(* IEC 61131-3 sources: RL_MAR/experiments/comparison/llm4plc/results/deepseek-ai-DeepSeek-V3.2_20260506_104945/20260506_124247, 4 files *)

(* ---- generated_code_iteration_0.st ---- *)
START_ST
FUNCTION_BLOCK MultimediaArtInstallationControl
VAR_INPUT
    MotionSensor : BOOL; (* Motion detection input *)
    AudioTrack : BOOL; (* Selected audio track *)
    VisualContent : BOOL; (* Selected visual content *)
END_VAR
VAR_OUTPUT
    LightingControl : BOOL; (* Lighting control output *)
    AudioControl : BOOL; (* Audio playback control *)
    VisualControl : BOOL; (* Visual display control *)
END_VAR
VAR
    ActivationTimer : INT; (* Timer for activation duration *)
    state : INT; (* Current state: 0 = IDLE_WAITING_FOR_MOTION, 1 = ACTIVE_ELEMENTS_ON *)
    prevState : INT; (* Previous state for detecting state changes *)
END_VAR

(* State definitions *)
CONST
    STATE_IDLE := 0;
    STATE_ACTIVE := 1;
END_CONST

(* State machine execution *)
CASE state OF
    STATE_IDLE: (* IDLE_WAITING_FOR_MOTION *)
        (* Set outputs to FALSE *)
        LightingControl := FALSE;
        AudioControl := FALSE;
        VisualControl := FALSE;

        (* Check transition to ACTIVE_ELEMENTS_ON *)
        IF MotionSensor THEN
            (* Reset timer and transition to active state *)
            ActivationTimer := 0;
            state := STATE_ACTIVE;
        END_IF;

    STATE_ACTIVE: (* ACTIVE_ELEMENTS_ON *)
        (* Set outputs to TRUE *)
        LightingControl := TRUE;
        AudioControl := TRUE;
        VisualControl := TRUE;

        (* Increment activation timer each cycle *)
        ActivationTimer := ActivationTimer + 1;

        (* Check transition back to IDLE *)
        IF (NOT MotionSensor) OR (ActivationTimer >= 300) THEN
            (* Reset timer and transition to idle state *)
            ActivationTimer := 0;
            state := STATE_IDLE;
        END_IF;

END_CASE;

(* Store current state for next cycle *)
prevState := state;

END_FUNCTION_BLOCK
END_ST

(* ---- generated_code_iteration_1.st ---- *)
START_REASON
The validation feedback indicates a syntax error in the CODESYS compiler validation. Specifically, it states: "应该用';' 替换'STATE_IDLE'", which translates to "should replace 'STATE_IDLE' with ';'". This suggests that in the CONST section, the constant declaration for STATE_IDLE is missing a semicolon at the end of the line. In Structured Text (ST), constant declarations must end with a semicolon, similar to variable declarations. The current code has "STATE_IDLE := 0;" but the feedback implies it's incorrectly written. However, looking at the provided code, the CONST section is:

CONST
    STATE_IDLE := 0;
    STATE_ACTIVE := 1;
END_CONST

This appears correct with semicolons. But the feedback might be pointing to a deeper issue: in CODESYS, constant declarations in a FUNCTION_BLOCK might require a different syntax or placement. Alternatively, the error could be due to a missing semicolon after "END_CONST" or an issue with the CASE statement. Upon review, the CASE statement uses "STATE_IDLE:" as a label, which is correct. The feedback might be misleading, but to comply, I'll ensure all syntax is correct. Perhaps the CONST section should be inside the VAR block or declared differently. In CODESYS, constants can be declared within the VAR_CONSTANT section. I'll restructure the code to use VAR_CONSTANT instead of CONST for better CODESYS compatibility. Also, I'll verify all semicolons are properly placed.

Additionally, I'll ensure the FUNCTION_BLOCK structure is maintained with proper variable sections closed with END_VAR, not END_VAR_INPUT or END_VAR_OUTPUT. The current code uses END_VAR correctly, but I'll double-check.

The core issue is likely the CONST declaration method. I'll change it to VAR_CONSTANT to align with CODESYS standards.
END_REASON

START_ST
FUNCTION_BLOCK MultimediaArtInstallationControl
VAR_INPUT
    MotionSensor : BOOL; (* Motion detection input *)
    AudioTrack : BOOL; (* Selected audio track *)
    VisualContent : BOOL; (* Selected visual content *)
END_VAR
VAR_OUTPUT
    LightingControl : BOOL; (* Lighting control output *)
    AudioControl : BOOL; (* Audio playback control *)
    VisualControl : BOOL; (* Visual display control *)
END_VAR
VAR
    ActivationTimer : INT; (* Timer for activation duration *)
    state : INT; (* Current state: 0 = IDLE_WAITING_FOR_MOTION, 1 = ACTIVE_ELEMENTS_ON *)
    prevState : INT; (* Previous state for detecting state changes *)
END_VAR
VAR_CONSTANT
    STATE_IDLE : INT := 0;
    STATE_ACTIVE : INT := 1;
END_VAR

(* State machine execution *)
CASE state OF
    STATE_IDLE: (* IDLE_WAITING_FOR_MOTION *)
        (* Set outputs to FALSE *)
        LightingControl := FALSE;
        AudioControl := FALSE;
        VisualControl := FALSE;

        (* Check transition to ACTIVE_ELEMENTS_ON *)
        IF MotionSensor THEN
            (* Reset timer and transition to active state *)
            ActivationTimer := 0;
            state := STATE_ACTIVE;
        END_IF;

    STATE_ACTIVE: (* ACTIVE_ELEMENTS_ON *)
        (* Set outputs to TRUE *)
        LightingControl := TRUE;
        AudioControl := TRUE;
        VisualControl := TRUE;

        (* Increment activation timer each cycle *)
        ActivationTimer := ActivationTimer + 1;

        (* Check transition back to IDLE *)
        IF (NOT MotionSensor) OR (ActivationTimer >= 300) THEN
            (* Reset timer and transition to idle state *)
            ActivationTimer := 0;
            state := STATE_IDLE;
        END_IF;

END_CASE;

(* Store current state for next cycle *)
prevState := state;

END_FUNCTION_BLOCK
END_ST

(* ---- generated_code_iteration_2.st ---- *)
START_REASON
The validation feedback indicates an encoding issue with the CODESYS compiler, specifically: "'gbk' codec can't decode byte 0xaf in position 129: illegal multibyte sequence". This suggests that there are non-ASCII characters in the code that the compiler cannot decode using the GBK encoding. The most likely source is the Chinese comments in the code, such as "(* Motion detection input *)" and others. CODESYS might be expecting ASCII-only characters or a different encoding. To fix this, I need to remove all non-ASCII characters from the code, including any Chinese or special characters in comments. I'll replace the Chinese comments with simple English comments or remove them entirely to ensure compatibility. Additionally, I'll ensure that all syntax is correct, using VAR_CONSTANT for constants and proper semicolon usage. The previous code already uses VAR_CONSTANT, but I'll verify there are no hidden non-ASCII characters. I'll rewrite the comments in plain English without special characters.
END_REASON

START_ST
FUNCTION_BLOCK MultimediaArtInstallationControl
VAR_INPUT
    MotionSensor : BOOL;
    AudioTrack : BOOL;
    VisualContent : BOOL;
END_VAR
VAR_OUTPUT
    LightingControl : BOOL;
    AudioControl : BOOL;
    VisualControl : BOOL;
END_VAR
VAR
    ActivationTimer : INT;
    state : INT;
    prevState : INT;
END_VAR
VAR_CONSTANT
    STATE_IDLE : INT := 0;
    STATE_ACTIVE : INT := 1;
END_VAR

CASE state OF
    STATE_IDLE:
        LightingControl := FALSE;
        AudioControl := FALSE;
        VisualControl := FALSE;

        IF MotionSensor THEN
            ActivationTimer := 0;
            state := STATE_ACTIVE;
        END_IF;

    STATE_ACTIVE:
        LightingControl := TRUE;
        AudioControl := TRUE;
        VisualControl := TRUE;

        ActivationTimer := ActivationTimer + 1;

        IF (NOT MotionSensor) OR (ActivationTimer >= 300) THEN
            ActivationTimer := 0;
            state := STATE_IDLE;
        END_IF;

END_CASE;

prevState := state;

END_FUNCTION_BLOCK
END_ST

(* ---- generated_code_iteration_3.st ---- *)
START_REASON
The CODESYS compiler validation failed because it requires VAR_CONSTANT to be replaced with VAR, VAR_INPUT, VAR_OUTPUT, or VAR_IN_OUT. In CODESYS Structured Text, constants should be declared within a VAR section using the CONSTANT keyword, not as a separate VAR_CONSTANT block. The correct syntax is to declare constants inside the VAR section with the CONSTANT attribute. I need to move the STATE_IDLE and STATE_ACTIVE constants into the VAR section and mark them as CONSTANT. This will resolve the compiler error. Additionally, I'll ensure all comments are in plain English to avoid encoding issues, though the previous feedback didn't mention that this time. I'll maintain the function block structure and use proper END_VAR closures.
END_REASON

START_ST
FUNCTION_BLOCK MultimediaArtInstallationControl
VAR_INPUT
    MotionSensor : BOOL;
    AudioTrack : BOOL;
    VisualContent : BOOL;
END_VAR
VAR_OUTPUT
    LightingControl : BOOL;
    AudioControl : BOOL;
    VisualControl : BOOL;
END_VAR
VAR
    ActivationTimer : INT;
    state : INT;
    prevState : INT;
    STATE_IDLE : INT := 0;
    STATE_ACTIVE : INT := 1;
END_VAR

CASE state OF
    STATE_IDLE:
        LightingControl := FALSE;
        AudioControl := FALSE;
        VisualControl := FALSE;

        IF MotionSensor THEN
            ActivationTimer := 0;
            state := STATE_ACTIVE;
        END_IF;

    STATE_ACTIVE:
        LightingControl := TRUE;
        AudioControl := TRUE;
        VisualControl := TRUE;

        ActivationTimer := ActivationTimer + 1;

        IF (NOT MotionSensor) OR (ActivationTimer >= 300) THEN
            ActivationTimer := 0;
            state := STATE_IDLE;
        END_IF;

END_CASE;

prevState := state;

END_FUNCTION_BLOCK
END_ST
